PROGRAM Atornillar_UR5
VAR
END_VAR

VAR_INPUT
	Iniciar : Bool;
	Corriente : REAL :=10;
	Vueltas : REAL := 1;
	giro_alivio : LREAL := 0;
END_VAR
VAR_OUTPUT
END_VAR
VAR
	cal_vueltas : REAL;
	ct : INT;
	TIME_IN :TIME := T#10000MS;
	wait_t : BOOL;
END_VAR

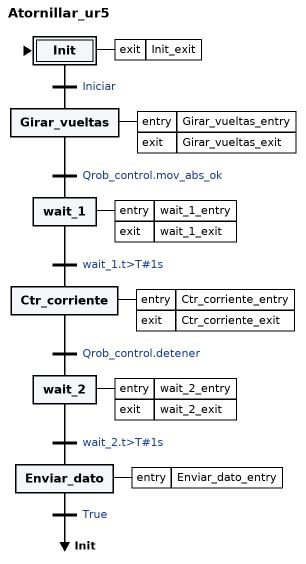
INITIAL_STEP Init:
    Init_exit(P0);  // exit action
END_STEP
TRANSITION FROM Init TO Girar_vueltas
    := Iniciar;
END_TRANSITION
STEP Girar_vueltas:
    Girar_vueltas_entry(P1);  // entry action
    Girar_vueltas_exit(P0);  // exit action
END_STEP
TRANSITION FROM Girar_vueltas TO wait_1
    := Qrob_control.mov_abs_ok;
END_TRANSITION
STEP wait_1:
    wait_1_entry(P1);  // entry action
    wait_1_exit(P0);  // exit action
END_STEP
TRANSITION FROM wait_1 TO Ctr_corriente
    := wait_1.t>T#1s;
END_TRANSITION
STEP Ctr_corriente:
    Ctr_corriente_entry(P1);  // entry action
    Ctr_corriente_exit(P0);  // exit action
END_STEP
TRANSITION FROM Ctr_corriente TO wait_2
    := Qrob_control.detener;
END_TRANSITION
STEP wait_2:
    wait_2_entry(P1);  // entry action
    wait_2_exit(P0);  // exit action
END_STEP
TRANSITION FROM wait_2 TO Enviar_dato
    := wait_2.t>T#1s;
END_TRANSITION
STEP Enviar_dato:
    Enviar_dato_entry(P1);  // entry action
END_STEP
TRANSITION FROM Enviar_dato TO Init
    := True;
END_TRANSITION

ACTION Alivio_torque_entry:
//regreo un grado para aliviar el torque y que pueda salir la herramienta
//Robot_A.UR_inputs.Bits.B11 := TRUE;
//wait_t := FALSE;
//Qrob_control.pos_mover_abs := Qrob_control.actual_position - giro_alivio;
//Qrob_control.velocidad := 50;
//Qrob_control.mover_abs := TRUE;


//Qrob_control.ajustar_tornillo := TRUE;
//Qrob_control.torque_relief := TRUE;
//Qrob_control.pos_mover_abs := Qrob_control.actual_position - giro_alivio;
//Qrob_control.velocidad := 0.5;
//Qrob_control.limite_corriente := 10;
//Qrob_control.mover_abs := TRUE;
END_ACTION

ACTION Alivio_torque_exit:

Robot_A.UR_inputs.Bits.B10 := FALSE;
//Qrob_control.ajustar_tornillo := FALSE;
//Qrob_control.torque_relief := FALSE;
Qrob_control.mover_abs := FALSE;
Qrob_control.detener := TRUE;
Qrob_control.detener := FALSE;
END_ACTION

ACTION Ctr_corriente_entry:
//cuando haya llegado al numero de vueltas especificado , realizo control de corriente 

wait_t := FALSE;
//FOR ct:=1 TO 5000 BY 1 DO
//Qrob_control.velocidad := 20;  
//END_FOR;

Qrob_control.ajustar_tornillo := TRUE;
Qrob_control.pos_mover_abs := 5000000;	
Qrob_control.velocidad := 100;
Qrob_control.limite_corriente := Corriente;
Qrob_control.mover_abs := TRUE;
END_ACTION

ACTION Ctr_corriente_exit:

Qrob_control.ajustar_tornillo := FALSE;
Qrob_control.detener := TRUE;
Qrob_control.detener := FALSE;
Qrob_control.mover_abs := FALSE;
END_ACTION

ACTION Enviar_dato_entry:

Robot_A.UR_inputs.Bits.B7 := TRUE;
Global_servo.Atornillado_ok :=TRUE;
END_ACTION

ACTION Girar_vueltas_entry:
// muevo ciertas cantidas d evuelatas a mayor velocidad y sin control de corriente 
Qrob_control.ajustar_tornillo := FALSE;


cal_vueltas := Qrob_control.actual_position + vueltas*360;
Qrob_control.pos_mover_abs := cal_vueltas;	
Qrob_control.velocidad := 180;
Qrob_control.mover_abs := TRUE;
END_ACTION

ACTION Girar_vueltas_exit:
Qrob_control.detener := TRUE;
Qrob_control.detener := FALSE;
Qrob_control.mover_abs := FALSE;
END_ACTION

ACTION Init_exit:

Robot_A.UR_inputs.Bits.B7 := FALSE;
Robot_A.UR_inputs.Bits.B8 := FALSE;
Iniciar := False;
END_ACTION

ACTION wait_1_entry:
Robot_A.UR_inputs.Bits.B10 := TRUE;
Qrob_control.detener := TRUE;
Qrob_control.detener := FALSE;
Qrob_control.mover_abs := FALSE;
END_ACTION

ACTION wait_1_exit:
Robot_A.UR_inputs.Bits.B10 := FALSE;
END_ACTION

ACTION wait_2_entry:


Qrob_control.detener := TRUE;
Qrob_control.detener := FALSE;
Qrob_control.mover_abs := FALSE;

Robot_A.UR_inputs.Bits.B7 := True;
END_ACTION

ACTION wait_2_exit:
Robot_A.UR_inputs.Bits.B7 := FALSE;
END_ACTION

END_PROGRAM

(* stored: Version 1.1.0.1, ProductVersion 3.1.4024.4
   POU Atornillar_ur5: Id {0d9be793-9cf9-44fe-8dfe-ac68b5df73fc}, SpecialFunc None
   Action Alivio_torque_entry: Id {ec2dcf41-5e2b-4524-895f-a6ff0483c002}
   Action Alivio_torque_exit: Id {64633a47-3658-49c4-83c7-e5bbedb36308}
   Action Ctr_corriente_entry: Id {68036340-2823-4b8d-b39a-dd07da0336bb}
   Action Ctr_corriente_exit: Id {39662e89-4599-463e-8fd7-b1c6ee3965f0}
   Action Enviar_dato_entry: Id {d8023a6b-cbe1-40ee-ac5f-a207eb6d2fcf}
   Action Girar_vueltas_entry: Id {57495244-5d46-4124-aba2-e7462e6c8478}
   Action Girar_vueltas_exit: Id {96a51748-7eb5-4114-ac23-f7ab51737ad0}
   Action Init_exit: Id {4eeb8cc2-9ddd-4456-b285-f1e02411c6aa}
   Action wait_1_entry: Id {6dd96752-8a7c-4775-8821-c58dcda5a48e}
   Action wait_1_exit: Id {272cbecc-0615-48f3-a23f-ddd2624b83ba}
   Action wait_2_entry: Id {73326cc6-fcad-433a-b7aa-6984c2635ad3}
   Action wait_2_exit: Id {4db9faa5-6b6d-46b1-9412-eeb31fd3663a} *)
